RoboDK station: dynamixel.rdk

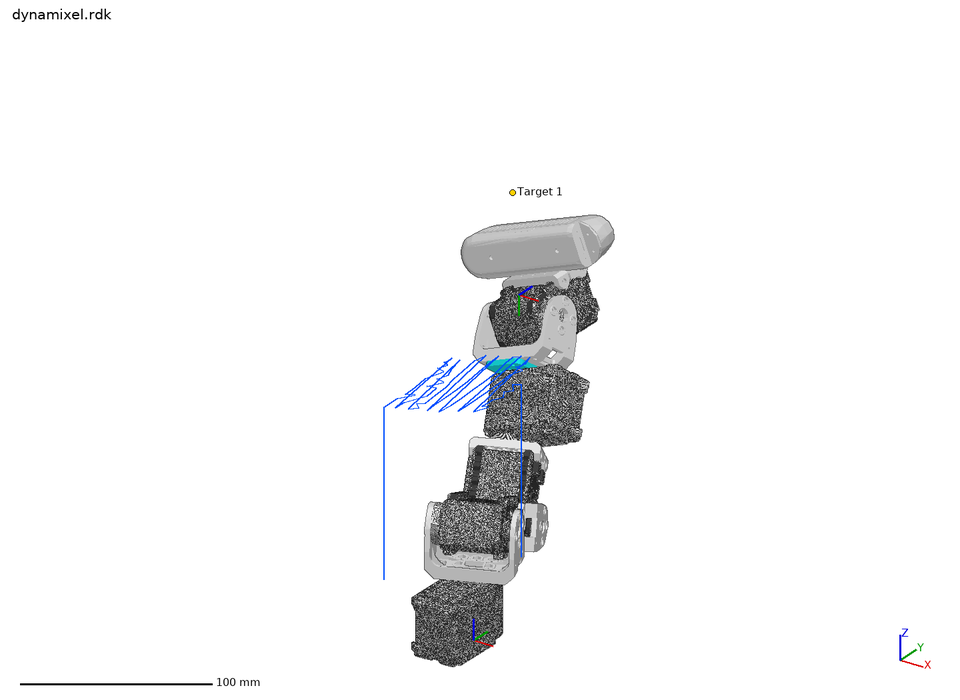
[picture v0: the station drawn from its stored meshes, robots at their saved joint values, targets as dots, program paths as lines]
Station dynamixel. Poses are relative to the parent item; angles as X-Y-Z fixed-axis rotations.
  - frame 我的机构 Base at (0, 2.24, 18.26) mm
    - robot : 6 axes
        modified DH rows (alpha deg, a mm, theta deg, d mm): 0, 0, 90, 66; -90, 0, -90, 0; 0, 67.5, 90, 0; -90, 0, 0, -111.8; 90, 0, 0, 0; -90, 0, 0, 0
        joint limits [-200, -200, -200, -200, -200, -200] to [200, 200, 200, 200, 200, 200]; home [0, 0, 0, 0, 0, 0]; saved at [23.223, 113.677, -70.142, 30.921, 50.112, -110.73]
      - tool Tool 1, TCP at (0, 0, 35) mm
    - target Target 1 (Cartesian target) at (0, 35, 245.3) mm, rotated rx 0 ry 90 rz 90 deg; joints [0, 0, 0, 0, 90, 0]
  - frame Object at (0, 43.03, 202.24) mm, rotated rx -89.34 ry 0 rz 0 deg
    - object Curve at (0, 0, 0) mm
  - machining project AutoCurveFollow settings: rotZ(0) | rotX(0)*rotY(0) | rotz(0) | onStart | onPathStart | onApproach | onPoint | onRetract | onFinish | SetRPM(%1) | SetTool(%1) | Extruder(%1) | default | default | OutOnMov(%1) | OutOffMov(%1) | onPathFinish | M_RunCode(%1)
  - program AutoCurveFollow (78 instructions, listed below)
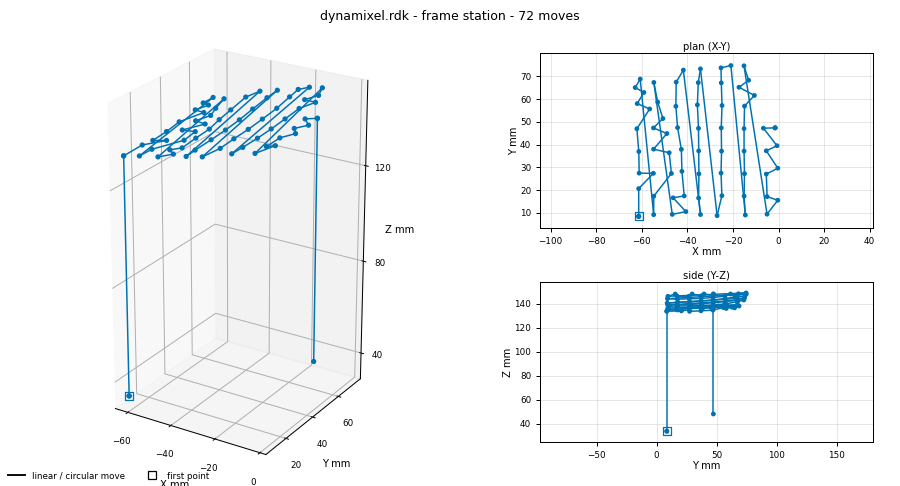
[picture p0: tool path of dynamixel.rdk in frame station, 72 of 72 moves have a stored position in this frame; points joined in program order, loops and branches not executed]

--- program AutoCurveFollow (robot ) ---
  Set Ref.: 我的机构 Base
  Set Tool: Tool 1
  Show Tool 1
  Set speed (1000.0 mm/s)
  MoveJ 1 to (-61.38, 6.26, 15.67) mm, rotated rx 0 ry 0 rz 180 deg; joints [70.673, 90.237, -91.497, 70.664, 89.758, -88.812]
  MoveL 2 to (-61.38, 6.26, 15.67) mm, rotated rx 0 ry 0 rz 180 deg; joints [70.673, 90.237, -91.497, 70.664, 89.758, -88.812]
  MoveL 3 to (-61.38, 6.26, 115.67) mm, rotated rx 0 ry 0 rz 180 deg; joints [26.797, 62.999, -20.173, 34.876, 52.037, -112.874]
  MoveL 4 to (-61.38, 6.26, 115.67) mm, rotated rx 0 ry 0 rz 180 deg; joints [26.797, 62.999, -20.173, 34.876, 52.037, -112.874]
  Set speed (5.0 mm/s)
  MoveL 5 to (-61.39, 18.44, 115.93) mm, rotated rx 0 ry 0 rz 180 deg; joints [26.724, 78.362, -39.338, 33.221, 55.16, -110.181]
  MoveL 6 to (-54.93, 25.15, 116.88) mm, rotated rx 0 ry 0 rz 180 deg; joints [24.074, 86.169, -49.151, 29.463, 56.024, -107.227]
  MoveL 7 to (-61.19, 25.23, 115.57) mm, rotated rx 0 ry 0 rz 180 deg; joints [26.705, 85.216, -47.173, 32.833, 55.976, -109.521]
  MoveL 8 to (-61.34, 34.72, 116) mm, rotated rx 0 ry 0 rz 180 deg; joints [26.658, 93.001, -54.692, 32.876, 55.737, -109.665]
  MoveL 9 to (-62.19, 44.72, 116.55) mm, rotated rx 0 ry 0 rz 180 deg; joints [26.852, 100.202, -60.608, 33.587, 54.729, -110.647]
  MoveL 10 to (-56.56, 53.39, 118.71) mm, rotated rx 0 ry 0 rz 180 deg; joints [24.328, 106.725, -66.197, 31.018, 53.072, -109.565]
  MoveL 11 to (-62.04, 55.76, 117.97) mm, rotated rx 0 ry 0 rz -180 deg; joints [26.507, 107.342, -65.506, 34.106, 52.741, -111.964]
  MoveL 12 to (-59.09, 60.63, 119) mm, rotated rx 0 ry 0 rz -180 deg; joints [25.217, 110.857, -68.296, 32.9, 51.659, -111.556]
  MoveL 13 to (-62.92, 62.8, 118.44) mm, rotated rx 0 ry 0 rz -180 deg; joints [26.728, 111.56, -67.948, 35.151, 51.365, -113.4]
  MoveL 14 to (-60.72, 66.51, 120) mm, rotated rx 0 ry 0 rz 180 deg; joints [25.632, 113.681, -69.052, 34.325, 50.095, -113.339]
  MoveL 15 to (-54.82, 6.99, 116.76) mm, rotated rx 0 ry 0 rz -180 deg; joints [24.086, 66.749, -26.458, 30.642, 53.194, -109.246]
  MoveL 16 to (-54.77, 15.11, 116.71) mm, rotated rx 0 ry 0 rz -180 deg; joints [24.061, 76.661, -38.777, 29.741, 55.267, -107.737]
  MoveL 17 to (-47.03, 25.09, 118.59) mm, rotated rx 0 ry 0 rz -180 deg; joints [20.671, 87.045, -50.976, 25.22, 55.936, -104.53]
  MoveL 18 to (-47.99, 34.18, 118.86) mm, rotated rx 0 ry 0 rz 180 deg; joints [20.999, 94.269, -57.696, 25.751, 55.565, -105.004]
  MoveL 19 to (-54.85, 35.75, 117.61) mm, rotated rx 0 ry 0 rz 180 deg; joints [23.897, 94.636, -57.087, 29.436, 55.509, -107.429]
  MoveL 20 to (-49.01, 42.61, 119) mm, rotated rx 0 ry 0 rz -180 deg; joints [21.369, 100.494, -62.938, 26.487, 54.78, -105.775]
  MoveL 21 to (-54.9, 45.08, 118.32) mm, rotated rx 0 ry 0 rz 180 deg; joints [23.775, 101.378, -62.616, 29.714, 54.417, -108.081]
  MoveL 22 to (-50.74, 49.19, 120) mm, rotated rx 0 ry 0 rz 180 deg; joints [21.882, 104.395, -65.12, 27.66, 53.395, -107.091]
  MoveL 23 to (-53.04, 56.4, 120.21) mm, rotated rx 0 ry 0 rz 180 deg; joints [22.727, 108.81, -67.773, 29.31, 52.106, -108.749]
  MoveL 24 to (-54.74, 65.03, 121.05) mm, rotated rx 0 ry 0 rz 180 deg; joints [23.223, 113.677, -70.142, 30.921, 50.112, -110.73]
  MoveL 25 to (-46.65, 7.13, 118.06) mm, rotated rx 0 ry 0 rz 180 deg; joints [20.631, 69.053, -30.7, 25.865, 53.865, -105.706]
  MoveL 26 to (-40.68, 8.36, 120) mm, rotated rx 0 ry 0 rz 180 deg; joints [17.908, 70.709, -32.876, 22.442, 53.651, -103.542]
  MoveL 27 to (-46.28, 14.4, 118.48) mm, rotated rx 0 ry 0 rz 180 deg; joints [20.401, 77.167, -40.389, 25.11, 55.226, -104.719]
  MoveL 28 to (-41.4, 15.23, 120) mm, rotated rx 0 ry 0 rz 180 deg; joints [18.194, 78.136, -41.621, 22.423, 54.936, -103.12]
  MoveL 29 to (-42.41, 26.04, 120.08) mm, rotated rx 0 ry 0 rz 180 deg; joints [18.582, 87.948, -51.993, 22.734, 55.542, -103.116]
  MoveL 30 to (-42.66, 35.66, 120.49) mm, rotated rx 0 ry 0 rz 180 deg; joints [18.611, 95.597, -59.106, 22.912, 55.054, -103.388]
  MoveL 31 to (-44.32, 45.2, 120.85) mm, rotated rx 0 ry 0 rz 180 deg; joints [19.218, 102.335, -64.411, 24.043, 53.885, -104.503]
  MoveL 32 to (-45.07, 54.57, 121.68) mm, rotated rx 0 ry 0 rz 180 deg; joints [19.386, 108.423, -68.501, 24.87, 52.11, -105.659]
  MoveL 33 to (-44.92, 65.18, 123.63) mm, rotated rx 0 ry 0 rz -180 deg; joints [19.039, 114.458, -71.46, 25.513, 49.229, -107.083]
  MoveL 34 to (-41.78, 70.45, 125) mm, rotated rx 0 ry 0 rz -180 deg; joints [17.616, 117.612, -73.191, 24.223, 47.525, -106.69]
  MoveL 35 to (-34.26, 7.06, 120.86) mm, rotated rx 0 ry 0 rz 180 deg; joints [15.127, 70.051, -32.705, 18.94, 53.508, -101.356]
  MoveL 36 to (-35.09, 14.3, 120.74) mm, rotated rx 0 ry 0 rz -180 deg; joints [15.483, 78.024, -42.209, 19.012, 55.025, -100.99]
  MoveL 37 to (-34.96, 24.93, 121.3) mm, rotated rx 0 ry 0 rz -180 deg; joints [15.347, 87.608, -52.288, 18.739, 55.468, -100.705]
  MoveL 38 to (-35.05, 34.99, 121.87) mm, rotated rx 0 ry 0 rz 180 deg; joints [15.308, 95.571, -59.656, 18.826, 54.897, -100.912]
  MoveL 39 to (-35.14, 44.9, 122.72) mm, rotated rx 0 ry 0 rz 180 deg; joints [15.234, 102.632, -65.265, 19.076, 53.509, -101.442]
  MoveL 40 to (-35.63, 55.2, 123.7) mm, rotated rx 0 ry 0 rz -180 deg; joints [15.316, 109.356, -69.782, 19.74, 51.445, -102.426]
  MoveL 41 to (-35.24, 64.95, 125.29) mm, rotated rx 0 ry 0 rz 180 deg; joints [14.967, 115.042, -72.707, 20.083, 48.771, -103.372]
  MoveL 42 to (-34.28, 70.99, 126.67) mm, rotated rx 0 ry 0 rz -180 deg; joints [14.425, 118.229, -73.896, 19.992, 46.766, -103.824]
  MoveL 43 to (-26.97, 6.59, 122.39) mm, rotated rx 0 ry 0 rz 180 deg; joints [11.878, 69.651, -32.342, 14.941, 52.97, -98.991]
  MoveL 44 to (-24.88, 15.33, 123.21) mm, rotated rx 0 ry 0 rz 180 deg; joints [10.901, 78.98, -43.254, 13.455, 54.361, -97.809]
  MoveL 45 to (-25.25, 25.25, 123.57) mm, rotated rx 0 ry 0 rz 180 deg; joints [11.02, 87.86, -52.546, 13.531, 54.778, -97.773]
  MoveL 46 to (-25.02, 34.89, 124.2) mm, rotated rx 0 ry 0 rz 180 deg; joints [10.862, 95.467, -59.558, 13.438, 54.178, -97.834]
  MoveL 47 to (-25.16, 45.09, 124.96) mm, rotated rx 0 ry 0 rz 180 deg; joints [10.849, 102.794, -65.446, 13.672, 52.777, -98.245]
  MoveL 48 to (-24.81, 54.92, 126.23) mm, rotated rx 0 ry 0 rz 180 deg; joints [10.594, 109.123, -69.59, 13.759, 50.617, -98.708]
  MoveL 49 to (-25.14, 64.86, 127.63) mm, rotated rx 0 ry 0 rz -180 deg; joints [10.613, 114.942, -72.611, 14.37, 47.906, -99.621]
  MoveL 50 to (-25.25, 71.44, 128.59) mm, rotated rx 0 ry 0 rz 180 deg; joints [10.58, 118.543, -74.137, 14.815, 45.892, -100.308]
  MoveL 51 to (-20.93, 72.46, 130) mm, rotated rx 0 ry 0 rz 180 deg; joints [8.709, 118.748, -73.769, 12.358, 45.026, -98.702]
  MoveL 52 to (-14.58, 6.84, 126.1) mm, rotated rx 0 ry 0 rz 180 deg; joints [6.306, 68.178, -29.351, 8.148, 50.796, -95.098]
  MoveL 53 to (-15.11, 15.14, 125.69) mm, rotated rx 0 ry 0 rz -180 deg; joints [6.548, 78.038, -41.559, 8.193, 53.14, -94.861]
  MoveL 54 to (-14.96, 24.99, 126.01) mm, rotated rx 0 ry 0 rz -180 deg; joints [6.461, 87.079, -51.206, 8.023, 53.734, -94.691]
  MoveL 55 to (-15.14, 34.91, 126.36) mm, rotated rx 0 ry 0 rz 180 deg; joints [6.517, 95.097, -58.809, 8.135, 53.326, -94.804]
  MoveL 56 to (-15.14, 44.78, 127.12) mm, rotated rx 0 ry 0 rz -180 deg; joints [6.476, 102.195, -64.544, 8.231, 51.974, -95.018]
  MoveL 57 to (-14.94, 54.66, 128.17) mm, rotated rx 0 ry 0 rz 180 deg; joints [6.334, 108.66, -68.937, 8.291, 49.91, -95.288]
  MoveL 58 to (-10.61, 59.33, 130) mm, rotated rx 0 ry 0 rz 180 deg; joints [4.446, 110.996, -69.65, 5.974, 48.149, -93.942]
  MoveL 59 to (-17.37, 62.92, 128.62) mm, rotated rx 0 ry 0 rz 180 deg; joints [7.327, 113.799, -72.025, 9.882, 47.988, -96.566]
  MoveL 60 to (-13.15, 65.98, 130.2) mm, rotated rx 0 ry 0 rz 180 deg; joints [5.493, 115.125, -72.119, 7.572, 46.583, -95.157]
  MoveL 61 to (-15.17, 72.34, 130.89) mm, rotated rx 0 ry 0 rz 180 deg; joints [6.296, 118.586, -73.58, 8.972, 44.684, -96.332]
  MoveL 62 to (-5.06, 7.22, 128.1) mm, rotated rx 0 ry 0 rz 180 deg; joints [2.163, 67.196, -27.213, 2.849, 49.393, -91.83]
  MoveL 63 to (-0.34, 13.33, 130) mm, rotated rx 0 ry 0 rz -180 deg; joints [0.142, 73.052, -33.385, 0.186, 49.674, -90.119]
  MoveL 64 to (-5.02, 14.92, 128.17) mm, rotated rx 0 ry 0 rz 180 deg; joints [2.143, 76.419, -38.568, 2.738, 51.521, -91.68]
  MoveL 65 to (-5.38, 24.81, 128.17) mm, rotated rx 0 ry 0 rz 180 deg; joints [2.296, 85.973, -49.15, 2.892, 52.553, -91.733]
  MoveL 66 to (-0.34, 27.4, 130) mm, rotated rx 0 ry 0 rz 180 deg; joints [0.142, 87.065, -49.161, 0.181, 51.437, -90.111]
  MoveL 67 to (-5.4, 35.03, 128.5) mm, rotated rx 0 ry 0 rz -180 deg; joints [2.295, 94.346, -57.217, 2.903, 52.247, -91.752]
  MoveL 68 to (-0.68, 37.25, 130) mm, rotated rx 0 ry 0 rz 180 deg; joints [0.284, 95.233, -57.129, 0.365, 51.238, -90.225]
  MoveL 69 to (-6.65, 44.95, 128.77) mm, rotated rx 0 ry 0 rz 180 deg; joints [2.819, 101.749, -63.544, 3.618, 51.191, -92.237]
  MoveL 70 to (-1.51, 45.1, 130) mm, rotated rx 0 ry 0 rz -180 deg; joints [0.635, 101.215, -62.388, 0.822, 50.517, -90.516]
  Set speed (1000.0 mm/s)
  MoveL 71 to (-1.51, 45.1, 130) mm, rotated rx 0 ry 0 rz -180 deg; joints [0.635, 101.215, -62.388, 0.822, 50.517, -90.516]
  MoveL 72 to (-1.51, 45.1, 30) mm, rotated rx 0 ry 0 rz 180 deg; joints [2.382, 123.42, -133.727, 2.416, 99.639, -89.568]
